// TIA Portal V20 export
DATA_BLOCK "Config"   // DB20
// stored: Access Published, MemoryReserve 100, Namespace Unit1.Em2
   VAR
      em : "LAF_typeEmConfiguration";   // Configuration of EM Parameters
      axis : Array[0.._.U1EM2_NO_OF_AXES] of DB_ANY;
      cmJROutPnPLeftSafetyPin : "LBC_typeDigitalSignalConfiguration";
      cmJROutPnPLeftJRDetect : "LBC_typeDigitalSignalConfiguration";
      cmJROutPnPRightSafetyPin : "LBC_typeDigitalSignalConfiguration";
      cmJROutPnPRightJRDetect : "LBC_typeDigitalSignalConfiguration";
   END_VAR
   VAR RETAIN
      cmJROutPnPLeftAxisX : "LBC_typeAxis64PosConfiguration";
      cmJROutPnPLeftAxisZ : "LBC_typeAxis64PosConfiguration";
      cmJROutPnPRightAxisX : "LBC_typeAxis64PosConfiguration";
      cmJROutPnPRightAxisZ : "LBC_typeAxis64PosConfiguration";
   END_VAR
   VAR
      cmJROutPnPLeftClampOpenClose : "LBC_typeTwoWayActuatorConfiguration";
      cmJROutPnPRightClampOpenClose : "LBC_typeTwoWayActuatorConfiguration";
      cmPowerMeter : "LER_typePAC3220Configuration";
      softcam : Struct
         JROutPnPLeftAxisX : "LER_typeSoftCamInterface";
         JROutPnPLeftAxisZ : "LER_typeSoftCamInterface";
         JROutPnPRightAxisX : "LER_typeSoftCamInterface";
         JROutPnPRightAxisZ { S7_SetPoint := 'True'} : "LER_typeSoftCamInterface";
      END_STRUCT;
   END_VAR
BEGIN
   em.referenceDesignator.parent := WSTRING#'U1';
   em.referenceDesignator.relative := WSTRING#'EM0';
   cmJROutPnPLeftAxisX.referenceDesignator := WSTRING#'OUT P&P LEFT X-Axis';
   cmJROutPnPLeftAxisX.setPositions[0].position := 4273.91;
   cmJROutPnPLeftAxisX.setPositions[1].position := -9.0;
   cmJROutPnPLeftAxisX.setPositions[2].position := 4273.91;
   cmJROutPnPLeftAxisX.setPositions[3].position := 4825.92;
   cmJROutPnPLeftAxisX.setPositions[0..3].velocity := 50.0;
   cmJROutPnPLeftAxisX.setPositions[0..3].acceleration := 500.0;
   cmJROutPnPLeftAxisX.setPositions[0..3].deceleration := 500.0;
   cmJROutPnPLeftAxisX.setPositions[0]."name" := 'Wait';
   cmJROutPnPLeftAxisX.setPositions[1]."name" := 'Stack1 Load';
   cmJROutPnPLeftAxisX.setPositions[2]."name" := 'Stack2 Load';
   cmJROutPnPLeftAxisX.setPositions[3]."name" := 'Unload';
   cmJROutPnPLeftAxisZ.referenceDesignator := WSTRING#'OUT P&P LEFT Z-Axis';
   cmJROutPnPLeftAxisZ.setPositions[0].position := 0.0;
   cmJROutPnPLeftAxisZ.setPositions[1..2].position := 356.0;
   cmJROutPnPLeftAxisZ.setPositions[3].position := 329.0;
   cmJROutPnPLeftAxisZ.setPositions[0..3].velocity := 10.0;
   cmJROutPnPLeftAxisZ.setPositions[0..3].acceleration := 100.0;
   cmJROutPnPLeftAxisZ.setPositions[0..3].deceleration := 100.0;
   cmJROutPnPLeftAxisZ.setPositions[0]."name" := 'Wait';
   cmJROutPnPLeftAxisZ.setPositions[1]."name" := 'Stack1 Load';
   cmJROutPnPLeftAxisZ.setPositions[2]."name" := 'Stack2 Load';
   cmJROutPnPLeftAxisZ.setPositions[3]."name" := 'Unload';
   cmJROutPnPRightAxisX.referenceDesignator := WSTRING#'OUT P&P RIGHT X-Axis';
   cmJROutPnPRightAxisX.setPositions[0].position := 600.0;
   cmJROutPnPRightAxisX.setPositions[1].position := 1277.8;
   cmJROutPnPRightAxisX.setPositions[2].position := 5.0;
   cmJROutPnPRightAxisX.setPositions[0..2].velocity := 50.0;
   cmJROutPnPRightAxisX.setPositions[0..2].acceleration := 500.0;
   cmJROutPnPRightAxisX.setPositions[0..2].deceleration := 500.0;
   cmJROutPnPRightAxisX.setPositions[0]."name" := 'Wait';
   cmJROutPnPRightAxisX.setPositions[1]."name" := 'Load';
   cmJROutPnPRightAxisX.setPositions[2]."name" := 'Unload';
   cmJROutPnPRightAxisZ.referenceDesignator := WSTRING#'OUT P&P RIGHT Z-Axis';
   cmJROutPnPRightAxisZ.setPositions[0..1].position := 16.86;
   cmJROutPnPRightAxisZ.setPositions[2].position := 480.0;
   cmJROutPnPRightAxisZ.setPositions[0..2].velocity := 10.0;
   cmJROutPnPRightAxisZ.setPositions[0..2].acceleration := 100.0;
   cmJROutPnPRightAxisZ.setPositions[0..2].deceleration := 100.0;
   cmJROutPnPRightAxisZ.setPositions[0]."name" := 'Wait';
   cmJROutPnPRightAxisZ.setPositions[1]."name" := 'Load';
   cmJROutPnPRightAxisZ.setPositions[2]."name" := 'Unload';
   cmJROutPnPLeftClampOpenClose.referenceDesignator := WSTRING#'OUT P&P LEFT GRIPPER';
   cmJROutPnPLeftClampOpenClose.monitoringDiscrepancy := T#5s;
   cmJROutPnPRightClampOpenClose.referenceDesignator := WSTRING#'OUT P&P RIGHT GRIPPER';
   cmJROutPnPRightClampOpenClose.monitoringDiscrepancy := T#5s;
   cmPowerMeter."Basic type 3_HW_ID" := 306;
END_DATA_BLOCK
